FUNCTION_BLOCK SS5_ps_Camera (* Composite FB wrapping other FBs *)
  (* Standard: 61499-2 *)
  (* Version 1.0, 2025-08-25, PS_Transformer_for_Unknown *)
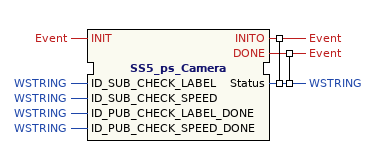
  EVENT_INPUT
    INIT; (* Initialization Request *)
  END_EVENT
  EVENT_OUTPUT
    INITO WITH Status; (* Initialization Confirm *)
    DONE WITH Status; (* Execution Confirmation *)
  END_EVENT
  VAR_INPUT
    ID_SUB_CHECK_LABEL : WSTRING;
    ID_SUB_CHECK_SPEED : WSTRING;
    ID_PUB_CHECK_LABEL_DONE : WSTRING;
    ID_PUB_CHECK_SPEED_DONE : WSTRING;
  END_VAR
  VAR_OUTPUT
    Status : WSTRING; (* Output event qualifier *)
  END_VAR
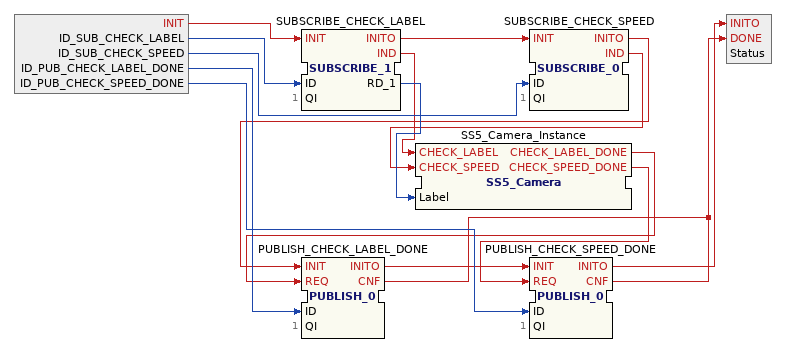
  FBS
    SS5_Camera_Instance : SS5_Camera;
    SUBSCRIBE_CHECK_LABEL : SUBSCRIBE_1(QI := 1);
    SUBSCRIBE_CHECK_SPEED : SUBSCRIBE_0(QI := 1);
    PUBLISH_CHECK_LABEL_DONE : PUBLISH_0(QI := 1);
    PUBLISH_CHECK_SPEED_DONE : PUBLISH_0(QI := 1);
  END_FBS
  EVENT_CONNECTIONS
    INIT TO SUBSCRIBE_CHECK_LABEL.INIT;
    SUBSCRIBE_CHECK_LABEL.INITO TO SUBSCRIBE_CHECK_SPEED.INIT;
    SUBSCRIBE_CHECK_SPEED.INITO TO PUBLISH_CHECK_LABEL_DONE.INIT;
    PUBLISH_CHECK_LABEL_DONE.INITO TO PUBLISH_CHECK_SPEED_DONE.INIT;
    PUBLISH_CHECK_SPEED_DONE.INITO TO INITO;
    SUBSCRIBE_CHECK_LABEL.IND TO SS5_Camera_Instance.CHECK_LABEL;
    SUBSCRIBE_CHECK_SPEED.IND TO SS5_Camera_Instance.CHECK_SPEED;
    SS5_Camera_Instance.CHECK_LABEL_DONE TO PUBLISH_CHECK_LABEL_DONE.REQ;
    SS5_Camera_Instance.CHECK_SPEED_DONE TO PUBLISH_CHECK_SPEED_DONE.REQ;
    PUBLISH_CHECK_LABEL_DONE.CNF TO DONE;
    PUBLISH_CHECK_SPEED_DONE.CNF TO DONE;
  END_CONNECTIONS
  DATA_CONNECTIONS
    ID_SUB_CHECK_LABEL TO SUBSCRIBE_CHECK_LABEL.ID;
    ID_SUB_CHECK_SPEED TO SUBSCRIBE_CHECK_SPEED.ID;
    ID_PUB_CHECK_LABEL_DONE TO PUBLISH_CHECK_LABEL_DONE.ID;
    ID_PUB_CHECK_SPEED_DONE TO PUBLISH_CHECK_SPEED_DONE.ID;
    SUBSCRIBE_CHECK_LABEL.RD_1 TO SS5_Camera_Instance.Label;
  END_CONNECTIONS
END_FUNCTION_BLOCK
